(*
SPDX-FileCopyrightText: © 2026 Oleksandr Tiutyk <trofimich@gmail.com>
SPDX-License-Identifier: MIT
License: https://opensource.org/license/mit
*)

{attribute 'no_explicit_call' := 'do not call this function block directly'} 
FUNCTION_BLOCK StringSplittingEnumerator EXTENDS Object IMPLEMENTS IEnumerator
VAR_OUTPUT
	SourceString : POINTER TO STRING;
	SourceStringLength : UDINT;
	SourceStringSize : UDINT;
	Separator : STRING;
	SeparatorLength : UDINT;
	MaxCount : UDINT := 0;
	TrimEntries : BOOL := FALSE;
	RemoveEmptyEntries : BOOL := FALSE;	
END_VAR
VAR
	{attribute 'hide'} 
	_ClassName : STRING := __POUNAME();

	{attribute 'hide'} 
	_CurrentString : POINTER TO STRING;
	{attribute 'hide'} 
	_CurrentStringLength : UDINT;
	{attribute 'hide'} 
	_CurrentEntry : POINTER TO STRING;
	{attribute 'hide'} 
	_CurrentEntrySize : UDINT;
	{attribute 'hide'} 
	_EntryCount : UDINT; 
END_VAR

{attribute 'monitoring' := 'call'}
PROPERTY ClassName : REFERENCE TO STRING
GET
ClassName REF= _ClassName;
END_GET
END_PROPERTY

(*!
<summary>Shows curent collection element</summary>
*)

{attribute 'monitoring' := 'call'}
PROPERTY Current : REFERENCE TO GENERIC_VALUE
GET
VAR_INST
	genericValue : GENERIC_VALUE;
END_VAR
IF _CurrentEntry <> 0 AND_THEN _CurrentEntrySize > 0 THEN
	genericValue := GenericValueFactory.FromParts(GENERIC_TYPE_CLASS.STRING_ASCII, _CurrentEntry, _CurrentEntrySize, GENERIC_MEMORY_MANAGEMENT_BEHAVIOR.STORE_ORIGINAL_REFERENCE_AND_NOT_OWNS_MEMORY);
ELSE
	genericValue.Reset();
END_IF

Current REF= genericValue;
END_GET
END_PROPERTY

PROPERTY CurrentEntry : REFERENCE TO STRING
GET
IF _CurrentEntry <> 0 THEN
	CurrentEntry REF= _CurrentEntry^;	
END_IF
END_GET
END_PROPERTY

//!<param name="bInCopyCode">if TRUE, the exit method is called for exiting an instance that is copied afterwards (online change).</param>

METHOD FB_exit : BOOL
VAR_INPUT
	
	bInCopyCode	: BOOL;
END_VAR
IF _CurrentEntry <> 0 THEN
	__DELETE(_CurrentEntry);
END_IF
END_METHOD

METHOD INTERNAL Initialize
VAR_INPUT
	sourceString : POINTER TO STRING;
END_VAR
VAR_IN_OUT CONSTANT
	separator : STRING;
END_VAR
VAR_INPUT
	maxCount : UDINT;
	trimEntries : BOOL;
	removeEmptyEntries : BOOL;
END_VAR
THIS^.SourceString := sourceString;
THIS^.SourceStringLength := Strings.InternalGetLength(sourceString);
THIS^.SourceStringSize := THIS^.SourceStringLength + Strings.CharSize; 
THIS^.Separator := separator;
THIS^.SeparatorLength := Strings.InternalGetLength(ADR(separator));
THIS^.MaxCount := maxCount;
THIS^.TrimEntries := trimEntries;
THIS^.RemoveEmptyEntries := removeEmptyEntries;

_CurrentString := THIS^.SourceString;

Reset();
END_METHOD

METHOD MoveNext : BOOL
VAR
	separatorPosition : UDINT;
END_VAR
START:

IF _CurrentEntry <> 0 THEN
	_CurrentEntrySize := 0;	
	__DELETE(_CurrentEntry);
END_IF

IF _CurrentString = 0 OR_ELSE _CurrentStringLength = 0 OR_ELSE Separator = '' OR_ELSE (MaxCount > 0 AND_THEN _EntryCount >= MaxCount) THEN
	RETURN;
END_IF

IF Strings.InternalFind(_CurrentString, _CurrentStringLength, ADR(Separator), SeparatorLength, position => separatorPosition) THEN
	_CurrentEntrySize := separatorPosition * Strings.CharSize;
	_CurrentEntry := __NEW(BYTE, _CurrentEntrySize);

	Tc2_System.MEMCPY(_CurrentEntry, _CurrentString, (separatorPosition - 1) * Strings.CharSize);
	Tc2_System.MEMSET(_CurrentEntry + ((separatorPosition - 1) * Strings.CharSize), 0, Strings.CharSize);

	_CurrentString := _CurrentString + ((separatorPosition - 1) * Strings.CharSize) + (SeparatorLength * Strings.CharSize);
	_CurrentStringLength := _CurrentStringLength - separatorPosition + 1 - SeparatorLength;
ELSE	
	_CurrentEntrySize := _CurrentStringLength + Strings.CharSize;	
	_CurrentEntry := __NEW(BYTE, _CurrentEntrySize);
	
	Tc2_System.MEMCPY(_CurrentEntry, _CurrentString, _CurrentStringLength + Strings.CharSize);
	
	_CurrentString := 0;
	_CurrentStringLength := 0;
END_IF

IF TrimEntries THEN
	Strings.TrimChar(_CurrentEntry^);
END_IF

IF RemoveEmptyEntries AND_THEN _CurrentEntry^ = '' THEN
	JMP START;
END_IF

_EntryCount := _EntryCount + 1;

MoveNext := TRUE;
END_METHOD

{attribute 'monitoring' := 'call'}
PROPERTY NamespaceName : REFERENCE TO STRING
GET
NamespaceName REF= CurrentNamespace.Name;
END_GET
END_PROPERTY

(*!
<summary>Releases the current fragment and resets iteration to before the first entry.</summary>
<description>
Preserves splitting settings and does not allocate memory or modify the source string.
Previously borrowed fragment addresses and references become invalid.
The initialized source string must remain alive and unchanged throughout iteration.
Repeated Reset calls are allowed, including before iteration and after its end.
</description>
*)
METHOD Reset
IF _CurrentEntry <> 0 THEN
	__DELETE(_CurrentEntry);
END_IF

_CurrentEntry := 0;
_CurrentEntrySize := 0;

_CurrentString := SourceString;
_CurrentStringLength := SourceStringLength;
_EntryCount := 0;
END_METHOD

{attribute 'monitoring' := 'call'}
PROPERTY SelfSize : ULINT
GET
SelfSize := XSIZEOF(THIS^);
END_GET
END_PROPERTY

END_FUNCTION_BLOCK

(* stored: Version 1.1.0.1
   POU StringSplittingEnumerator: Id {39677a7e-6822-49fb-a976-fd077aac311a}, SpecialFunc None
   Property ClassName: Id {dc8168cb-a7bf-4d33-9f6c-41b2c6a729dd}
   Get Get: Id {451b3de0-abf2-482f-a7cd-159e1ec34840}
   Property Current: Id {578ddaf1-4d15-456a-9c92-6ba01ccaf901}
   Get Get: Id {ff624da2-e0ce-48f6-a18a-67e4fe74d3a7}
   Property CurrentEntry: Id {3c87ffb4-1d5d-46d7-8e98-8f42eb9deaf3}
   Get Get: Id {df9fd113-3b9b-4abf-a069-25f1abcf0162}
   Method FB_exit: Id {91c3c83f-b495-4483-9409-84eb69a852b9}
   Method Initialize: Id {dd46f3d0-2251-42fe-acf7-cf970e2b2bc6}
   Method MoveNext: Id {b4c28f78-8b1f-47b3-af5b-cb333bb9b6f3}
   Property NamespaceName: Id {eac5bc76-1c0c-415a-b31e-3c5597f64aa3}
   Get Get: Id {2b679829-e2da-4785-aab9-24372420e1f5}
   Method Reset: Id {0c911c06-568e-4235-8bc3-600486eb4862}
   Property SelfSize: Id {07711580-08e7-4949-b5a3-b486d7b73972}
   Get Get: Id {80ff0b12-faeb-4d39-a7b6-5a5f5617c0d6} *)
